FUNCTION_BLOCK VALUES2ARRAY_2_LREAL
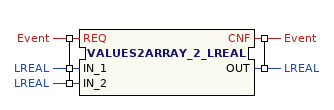
  EVENT_INPUT
    REQ WITH IN_1, IN_2;
  END_EVENT
  EVENT_OUTPUT
    CNF WITH OUT;
  END_EVENT
  VAR_INPUT
    IN_1 : LREAL;
    IN_2 : LREAL;
  END_VAR
  VAR_OUTPUT
    OUT : LREAL;
  END_VAR
END_FUNCTION_BLOCK
